SYSTEM Test System
  (* Version 1.0, 2005-06-15, Goran Cengic, Chalmers *)
  DEVICE Test Device : DeviceType_not_used
    RESOURCE TestResource : ResourceType_not_used
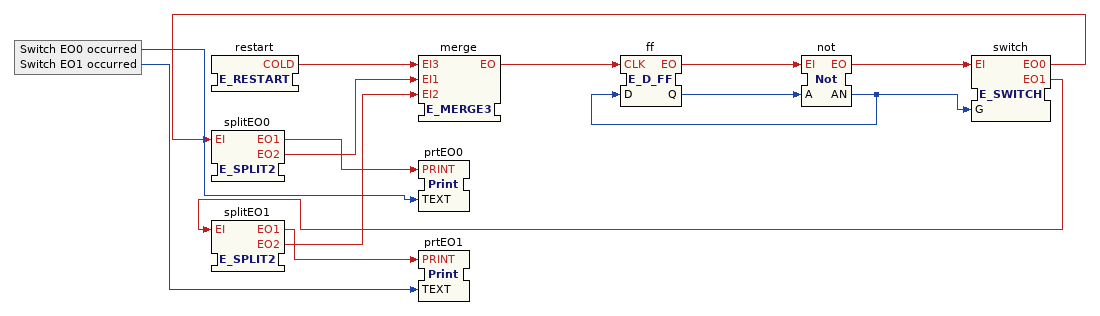
      FBS
        restart : E_RESTART;
        merge : E_MERGE3;
        splitEO0 : E_SPLIT2;
        splitEO1 : E_SPLIT2;
        ff : E_D_FF;
        not : Not;
        switch : E_SWITCH;
        prtEO0 : Print;
        prtEO1 : Print;
      END_FBS
      EVENT_CONNECTIONS
        restart.COLD TO merge.EI3;
        merge.EO TO ff.CLK;
        ff.EO TO not.EI;
        not.EO TO switch.EI;
        switch.EO0 TO splitEO0.EI;
        switch.EO1 TO splitEO1.EI;
        splitEO0.EO1 TO prtEO0.PRINT;
        splitEO1.EO1 TO prtEO1.PRINT;
        splitEO0.EO2 TO merge.EI1;
        splitEO1.EO2 TO merge.EI2;
      END_CONNECTIONS
      DATA_CONNECTIONS
        Switch EO0 occurred TO prtEO0.TEXT;
        Switch EO1 occurred TO prtEO1.TEXT;
        ff.Q TO not.A;
        not.AN TO switch.G;
        not.AN TO ff.D;
      END_CONNECTIONS
    END_RESOURCE
  END_DEVICE
END_SYSTEM
